# EPICS IOC start-up script: iocsh/iocStats-ioc.iocsh
dbLoadRecords("iocAdminSoft-freia-proc.db", "IOC=$(IOCNAME)")
